// TIA Portal V19 export
FUNCTION "FC_TransferDataPLC_LJX8000" : Void   // FC4, LAD
{ S7_Optimized_Access := 'TRUE' }
// stored: SetENOAutomatically false
BEGIN

REGION Network 1: PLC to LJ_X8000 bits
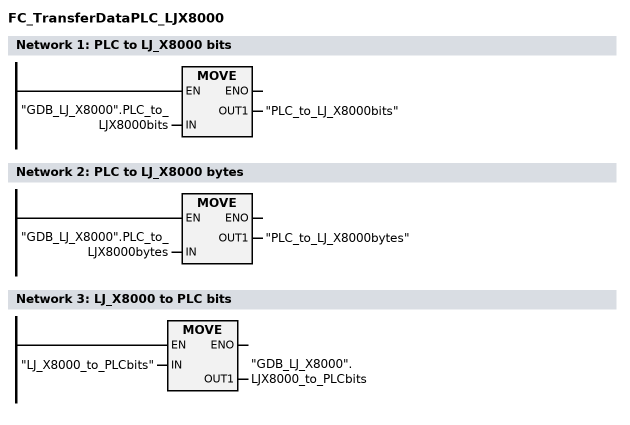
   RUNG wire#powerrail
      Move(in := "GDB_LJ_X8000".PLC_to_LJX8000bits, out1 => "PLC_to_LJ_X8000bits")
   END_RUNG
   // the same network as SCL:
   "PLC_to_LJ_X8000bits" := "GDB_LJ_X8000".PLC_to_LJX8000bits;
END_REGION

REGION Network 2: PLC to LJ_X8000 bytes
   RUNG wire#powerrail
      Move(in := "GDB_LJ_X8000".PLC_to_LJX8000bytes, out1 => "PLC_to_LJ_X8000bytes")
   END_RUNG
   // the same network as SCL:
   "PLC_to_LJ_X8000bytes" := "GDB_LJ_X8000".PLC_to_LJX8000bytes;
END_REGION

REGION Network 3: LJ_X8000 to PLC bits
   RUNG wire#powerrail
      Move(in := "LJ_X8000_to_PLCbits", out1 => "GDB_LJ_X8000".LJX8000_to_PLCbits)
   END_RUNG
   // the same network as SCL:
   "GDB_LJ_X8000".LJX8000_to_PLCbits := "LJ_X8000_to_PLCbits";
END_REGION
END_FUNCTION
